Staubli VAL3: RobotController.pjx

--- RobotController.pjx ---
Parameters version=s7.9.1 stackSize=5000 millimeterUnit=true
Program file=start.pgx
Program file=stop.pgx
Data file=RobotController.dtx
Library alias=connectHostRos path=./realtimeComm/connectHostRos/connectHostRos.pjx
Library alias=acqSensorData path=./realtimeComm/acqSensorData/acqSensorData.pjx
Library alias=exceptionHandle path=./exceptionHandle/exceptionHandle.pjx
Library alias=newMoveCmd path=./motionControl/newMoveCmd/newMoveCmd.pjx
Library alias=robotMove path=./motionControl/robotMove/robotMove.pjx
Library alias=robotPlanner path=./motionControl/robotPlanner/robotPlanner.pjx
Library alias=robotStatusInq path=./motionControl/robotStatusInq/robotStatusInq.pjx
Library alias=modelParmIdent path=./motionControl/modelParmIdent/modelParmIdent.pjx
Type name=FlagStatus path=Disk://RobotController_Libs/FlagStatus/FlagStatus.pjx

--- RobotController.dtx ---
mdesc mNomSpeed
public string sMotionTaskName
public string sScreenTaskName
public string sDataTaskName
public string sExceptTaskName
public string sCommTaskName
public string sMotionSocket
public string sFbkSocket
public FlagStatus fFlagStatus
  [0]
    num ForceFlag
    num RosFlag
    num RobotFlag
